INTERFACE ITF_Group3_HMI_Connector_View EXTENDS ITF_BaseGroupElement_HMI_Connector_View

END_INTERFACE

(* stored: Version 1.1.0.1
   Itf ITF_Group3_HMI_Connector_View: Id {7d5088e5-42b3-07d4-1015-89bd172ef654} *)
